PROGRAM MAIN
VAR
	Machine: FB_UM_Machine	:= (Name := 'Machine', LogStateChanges := TRUE);
	Initialized: BOOL;
END_VAR

CyclicLogic();

METHOD CyclicLogic : BOOL
VAR_INPUT
END_VAR
IF NOT Initialized THEN
    Initialized := Initialize();
    RETURN;
END_IF

Machine.CyclicLogic();
END_METHOD

METHOD Initialize : BOOL
VAR_INPUT
END_VAR
Initialize := TRUE;
END_METHOD

END_PROGRAM

(* stored: Version 1.1.0.1, ProductVersion 3.1.4024.12
   POU MAIN: Id {312512fd-d160-4e78-97b1-763f6b70b1ed}, SpecialFunc None
   Method CyclicLogic: Id {fe332985-0e52-4a1e-a556-33a8822260d7}
   Method Initialize: Id {b3cc5d6e-29f4-4149-9705-156e78b671c1} *)
